ABB RobotStudio station: CubesMovement_20241125-185710.rsstn

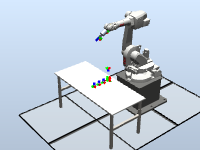
Station CubesMovement (saved by RobotStudio 6.8.8307.1040)
Controller System1, task T_ROB1: task frame (RAPID world) sits at (0, 0, 520) mm in the station
Controller System1
  mechanical unit ROB_1: IRB1600_10_145__01, 6 joints, base frame (0, 0, 0) mm
Layout (positions relative to the parent item):
  - IRB1600_10_145__01 [mechanism, from Robots\IRB1600_10_145_G_01.rslib] at (0, 0, 520) mm; joint values [0, 0, 0, 0, 0.5236, 0] (rad or m)
  - base [part, from Desktop\подставка.rslib]
  - table [part, from Desktop\Стол сборка.rslib] at (677.65, -723.32, 0) mm, rotated rx 0 ry 0 rz 90 deg
  - toolGripper [mechanism, from Desktop\toolGripper.rslib] at (806.29, 0, 1674) mm, rotated rx -180 ry 60 rz -180 deg
  - cube_1 [part, from Desktop\cube.rslib] at (844.98, -5.05, 730.16) mm
  - cube_2 [part, from Desktop\cube.rslib] at (944.98, -5.05, 730.39) mm
  - cube_3 [part, from Desktop\cube.rslib] at (1044.98, -5.05, 730.61) mm
Attachment: wobjTable is attached to table
Attachment: toolGripper is attached to IRB1600_10_145__01 / Link6
Collision set CollisionSet_1: IRB1600_10_145__01, toolGripper, table against table, toolGripper, near miss 0 m
EventTableEntry 1490: Group=, Trigger=close_cube_1_f 1624, Actions=[EventTableActionAttach 1492], Comment=, ActivationMode=2, Cyclic=false
EventTableActionAttach 1492: AttachmentParent=toolGripper 991, AttachmentChild=cube_1 995, MountObject=false, Offset=[X=1, Y=0, Z=0, W=0, X=0, Y=1, Z=0, W=0, X=0, Y=0, Z=1, W=0, X=0, Y=0, Z=0, W=1], FlangeIndext=0, FindNearest=false
EventTableEntry 1493: Group=, Trigger=open_cube_1_f 1625, Actions=[EventTableActionDetach 1495], Comment=, ActivationMode=2, Cyclic=false
EventTableActionDetach 1495: AttachmentParent=toolGripper 991, AttachmentChild=cube_1 995
EventTableEntry 1496: Group=, Trigger=close_cube_2_f 1626, Actions=[EventTableActionAttach 1498], Comment=, ActivationMode=2, Cyclic=false
EventTableActionAttach 1498: AttachmentParent=toolGripper 991, AttachmentChild=cube_2 996, MountObject=false, Offset=[X=1, Y=0, Z=0, W=0, X=0, Y=1, Z=0, W=0, X=0, Y=0, Z=1, W=0, X=0, Y=0, Z=0, W=1], FlangeIndext=0, FindNearest=false
EventTableEntry 1499: Group=, Trigger=open_cube_2_f 1627, Actions=[EventTableActionDetach 1501], Comment=, ActivationMode=2, Cyclic=false
EventTableActionDetach 1501: AttachmentParent=toolGripper 991, AttachmentChild=cube_2 996
EventTableEntry 1502: Group=, Trigger=close_cube_3_f 1628, Actions=[EventTableActionAttach 1504], Comment=, ActivationMode=2, Cyclic=false
EventTableActionAttach 1504: AttachmentParent=toolGripper 991, AttachmentChild=cube_3 997, MountObject=false, Offset=[X=1, Y=0, Z=0, W=0, X=0, Y=1, Z=0, W=0, X=0, Y=0, Z=1, W=0, X=0, Y=0, Z=0, W=1], FlangeIndext=0, FindNearest=false
EventTableEntry 1505: Group=, Trigger=open_cube_3_f 1629, Actions=[EventTableActionDetach 1507], Comment=, ActivationMode=2, Cyclic=false
EventTableActionDetach 1507: AttachmentParent=toolGripper 991, AttachmentChild=cube_3 997
EventTableEntry 1508: Group=, Trigger=close_cube_3_b 1630, Actions=[EventTableActionAttach 1510], Comment=, ActivationMode=2, Cyclic=false
EventTableActionAttach 1510: AttachmentParent=toolGripper 991, AttachmentChild=cube_3 997, MountObject=false, Offset=[X=1, Y=0, Z=0, W=0, X=0, Y=1, Z=0, W=0, X=0, Y=0, Z=1, W=0, X=0, Y=0, Z=0, W=1], FlangeIndext=0, FindNearest=false
EventTableEntry 1511: Group=, Trigger=open_cube_3_b 1631, Actions=[EventTableActionDetach 1513], Comment=, ActivationMode=2, Cyclic=false
EventTableActionDetach 1513: AttachmentParent=toolGripper 991, AttachmentChild=cube_3 997
EventTableTriggerIO 1624: IOValue=[1], IRC5Controller=? -1, Operator=0, SignalSource=System1 491
EventTableTriggerIO 1625: IOValue=[1], IRC5Controller=? -1, Operator=0, SignalSource=System1 491
EventTableTriggerIO 1626: IOValue=[1], IRC5Controller=? -1, Operator=0, SignalSource=System1 491
EventTableTriggerIO 1627: IOValue=[1], IRC5Controller=? -1, Operator=0, SignalSource=System1 491
EventTableTriggerIO 1628: IOValue=[1], IRC5Controller=? -1, Operator=0, SignalSource=System1 491
EventTableTriggerIO 1629: IOValue=[1], IRC5Controller=? -1, Operator=0, SignalSource=System1 491
EventTableTriggerIO 1630: IOValue=[1], IRC5Controller=? -1, Operator=0, SignalSource=System1 491
EventTableTriggerIO 1631: IOValue=[1], IRC5Controller=? -1, Operator=0, SignalSource=System1 491
EventTableEntry 1632: Group=, Trigger=close_cube_2_b 1633, Actions=[EventTableActionAttach 1634], Comment=, ActivationMode=2, Cyclic=false
EventTableTriggerIO 1633: IOValue=[1], IRC5Controller=? -1, Operator=0, SignalSource=System1 491
EventTableActionAttach 1634: AttachmentParent=toolGripper 991, AttachmentChild=cube_2 996, MountObject=false, Offset=[X=1, Y=0, Z=0, W=0, X=0, Y=1, Z=0, W=0, X=0, Y=0, Z=1, W=0, X=0, Y=0, Z=0, W=1], FlangeIndext=0, FindNearest=false
EventTableEntry 1635: Group=, Trigger=open_cube_2_b 1636, Actions=[EventTableActionDetach 1637], Comment=, ActivationMode=2, Cyclic=false
EventTableTriggerIO 1636: IOValue=[1], IRC5Controller=? -1, Operator=0, SignalSource=System1 491
EventTableActionDetach 1637: AttachmentParent=toolGripper 991, AttachmentChild=cube_2 996
EventTableEntry 1638: Group=, Trigger=close_cube_1_b 1639, Actions=[EventTableActionAttach 1640], Comment=, ActivationMode=2, Cyclic=false
EventTableTriggerIO 1639: IOValue=[1], IRC5Controller=? -1, Operator=0, SignalSource=System1 491
EventTableActionAttach 1640: AttachmentParent=toolGripper 991, AttachmentChild=cube_1 995, MountObject=false, Offset=[X=1, Y=0, Z=0, W=0, X=0, Y=1, Z=0, W=0, X=0, Y=0, Z=1, W=0, X=0, Y=0, Z=0, W=1], FlangeIndext=0, FindNearest=false
EventTableEntry 1641: Group=, Trigger=open_cube_1_b 1642, Actions=[EventTableActionDetach 1643], Comment=, ActivationMode=2, Cyclic=false
EventTableTriggerIO 1642: IOValue=[1], IRC5Controller=? -1, Operator=0, SignalSource=System1 491
EventTableActionDetach 1643: AttachmentParent=toolGripper 991, AttachmentChild=cube_1 995
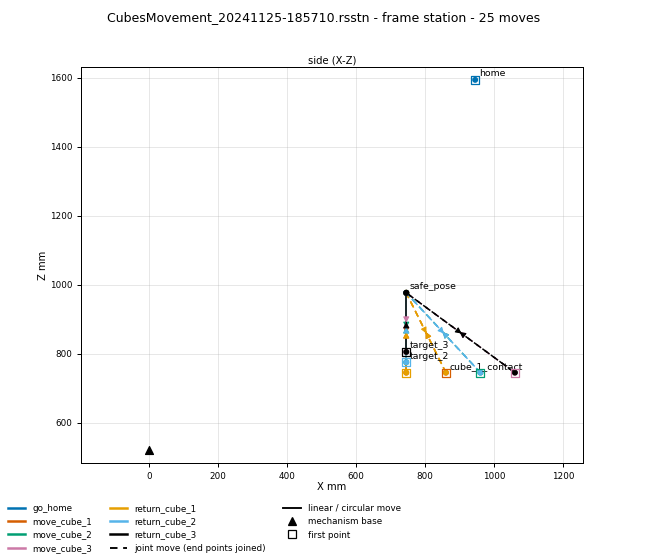
[picture p0: tool path of CubesMovement_20241125-185710.rsstn in frame station, 25 of 25 moves have a stored position in this frame; points joined in program order, loops and branches not executed]
Targets, tools, work objects and paths stored in the station, written as RAPID:
! task T_ROB1
MODULE CalibData
  PERS tooldata toolGripper:=[TRUE,[[0,0,160],[1,0,0,0]],[0.8,[0,0,1],[1,0,0,0],0,0,0]];
  TASK PERS wobjdata wobjTable:=[FALSE,TRUE,"",[[744.979,-5.048,210.071],[1,0,0,0]],[[0,0,0],[1,0,0,0]]];
ENDMODULE

! task T_ROB1
MODULE Module1
  CONST robtarget home:=[[944.855715851,0,1074],[0.5,0,0.866025404,0],[0,0,0,0],[9E+09,9E+09,9E+09,9E+09,9E+09,9E+09]];
  CONST robtarget cube_1_pose:=[[100,0,0],[1,0,0,0],[0,0,0,0],[9E+09,9E+09,9E+09,9E+09,9E+09,9E+09]];
  CONST robtarget cube_2_pose:=[[200,0,0],[1,0,0,0],[0,0,0,0],[9E+09,9E+09,9E+09,9E+09,9E+09,9E+09]];
  CONST robtarget cube_3_pose:=[[300,0,0],[1,0,0,0],[0,0,0,0],[9E+09,9E+09,9E+09,9E+09,9E+09,9E+09]];
  CONST robtarget tower_pose:=[[0,0,0],[1,0,0,0],[0,0,0,0],[9E+09,9E+09,9E+09,9E+09,9E+09,9E+09]];
  CONST robtarget cube_1_contact:=[[115,15,15],[0,0.707106781,0.707106781,0],[0,0,0,0],[9E+09,9E+09,9E+09,9E+09,9E+09,9E+09]];
  CONST robtarget cube_2_contact:=[[215,15,15],[0,0.707106781,0.707106781,0],[0,0,0,0],[9E+09,9E+09,9E+09,9E+09,9E+09,9E+09]];
  CONST robtarget cube_3_contact:=[[315,15,15],[0,0.707106781,0.707106781,0],[0,0,0,0],[9E+09,9E+09,9E+09,9E+09,9E+09,9E+09]];
  CONST robtarget target_1:=[[0,15,15],[0,0.707106781,0.707106781,0],[0,0,0,0],[9E+09,9E+09,9E+09,9E+09,9E+09,9E+09]];
  CONST robtarget target_2:=[[0,15,45],[0,0.707106781,0.707106781,0],[0,0,0,0],[9E+09,9E+09,9E+09,9E+09,9E+09,9E+09]];
  CONST robtarget target_3:=[[0,15,75],[0,0.707106781,0.707106781,0],[0,0,0,0],[9E+09,9E+09,9E+09,9E+09,9E+09,9E+09]];
  CONST robtarget safe_pose:=[[0.000003222,0.000000245,246.376418077],[0,0.707106781,0.707106781,0],[-1,-1,0,0],[9E+09,9E+09,9E+09,9E+09,9E+09,9E+09]];
  PROC go_home()
    MoveJ home,v100,fine,toolGripper\WObj:=wobj0;
  ENDPROC
  PROC main()
    go_home;
    move_cube_1;
    move_cube_2;
    move_cube_3;
    wait;
    return_cube_3;
    return_cube_2;
    return_cube_1;
    go_home;
  ENDPROC
  PROC move_cube_1()
    MoveJ cube_1_contact,v100,fine,toolGripper\WObj:=wobjTable;
    PulseDO \High,do_GripClose;
    PulseDO \High,close_cube_1_f;
    WaitTime 1;
    MoveJ safe_pose,v100,fine,toolGripper\WObj:=wobjTable;
    MoveL target_1,v100,fine,toolGripper\WObj:=wobjTable;
    PulseDO \High,do_GripOpen;
    PulseDO \High,open_cube_1_f;
    WaitTime 1;
    MoveL safe_pose,v100,fine,toolGripper\WObj:=wobjTable;
  ENDPROC
  PROC move_cube_2()
    MoveJ cube_2_contact,v100,fine,toolGripper\WObj:=wobjTable;
    PulseDO \High,do_GripClose;
    PulseDO \High,close_cube_2_f;
    WaitTime 1;
    MoveJ safe_pose,v100,fine,toolGripper\WObj:=wobjTable;
    MoveL target_2,v100,fine,toolGripper\WObj:=wobjTable;
    PulseDO \High,do_GripOpen;
    PulseDO open_cube_2_f;
    WaitTime 1;
    MoveL safe_pose,v100,fine,toolGripper\WObj:=wobjTable;
  ENDPROC
  PROC move_cube_3()
    MoveJ cube_3_contact,v100,fine,toolGripper\WObj:=wobjTable;
    PulseDO \High,do_GripClose;
    PulseDO \High,close_cube_3_f;
    WaitTime 1;
    MoveJ safe_pose,v100,fine,toolGripper\WObj:=wobjTable;
    MoveL target_3,v100,fine,toolGripper\WObj:=wobjTable;
    PulseDO \High,do_GripOpen;
    PulseDO \High,open_cube_3_f;
    WaitTime 1;
    MoveL safe_pose,v100,fine,toolGripper\WObj:=wobjTable;
  ENDPROC
  PROC return_cube_1()
    MoveL target_1,v100,fine,toolGripper\WObj:=wobjTable;
    PulseDO \High,do_GripClose;
    PulseDO \High,close_cube_1_b;
    WaitTime 1;
    MoveL safe_pose,v100,fine,toolGripper\WObj:=wobjTable;
    MoveJ cube_1_contact,v100,fine,toolGripper\WObj:=wobjTable;
    PulseDO \High,do_GripOpen;
    PulseDO \High,open_cube_1_b;
    WaitTime 1;
    MoveJ safe_pose,v100,fine,toolGripper\WObj:=wobjTable;
  ENDPROC
  PROC return_cube_2()
    MoveL target_2,v100,fine,toolGripper\WObj:=wobjTable;
    PulseDO \High,do_GripClose;
    PulseDO \High,close_cube_2_b;
    WaitTime 1;
    MoveL safe_pose,v100,fine,toolGripper\WObj:=wobjTable;
    MoveJ cube_2_contact,v100,fine,toolGripper\WObj:=wobjTable;
    PulseDO \High,do_GripOpen;
    PulseDO \High,open_cube_2_b;
    WaitTime 1;
    MoveJ safe_pose,v100,fine,toolGripper\WObj:=wobjTable;
  ENDPROC
  PROC return_cube_3()
    MoveL target_3,v100,fine,toolGripper\WObj:=wobjTable;
    PulseDO \High,do_GripClose;
    PulseDO \High,close_cube_3_b;
    WaitTime 1;
    MoveL safe_pose,v100,fine,toolGripper\WObj:=wobjTable;
    MoveJ cube_3_contact,v100,fine,toolGripper\WObj:=wobjTable;
    PulseDO \High,do_GripOpen;
    PulseDO open_cube_3_b;
    WaitTime 1;
    MoveJ safe_pose,v100,fine,toolGripper\WObj:=wobjTable;
  ENDPROC
  PROC wait()
    WaitTime 2;
  ENDPROC
ENDMODULE

